// TIA Portal V16 program export: 1 tag tables, 0 data types, 0 data blocks, 1 code blocks (in call order from the OBs), 0 instance data blocks

VAR_GLOBAL   // PLC tag table "Electrical_interlock tag table"
   Stop AT %I0.0 : Bool;
   Start AT %I0.1 : Bool;
   Sistem AT %Q0.0 : Bool;
   btn_ileri AT %I0.2 : Bool;
   m_ileri AT %Q0.1 : Bool;
   btn_geri AT %I0.3 : Bool;
   m_geri AT %Q0.2 : Bool;
END_VAR

ORGANIZATION_BLOCK "Electrical_interlock"   // OB1, LAD, ProgramCycle
TITLE = "Main Program Sweep (Cycle)"
{ S7_Optimized_Access := 'TRUE' }
VERSION : 0.1
// stored: AutoNumber true, IsIECCheckEnabled false, SetENOAutomatically false
   VAR_INPUT
      Initial_Call : Bool;   // Initial call of this OB
      Remanence : Bool;   // =True, if remanent data are available
   END_VAR
BEGIN

REGION Network 1
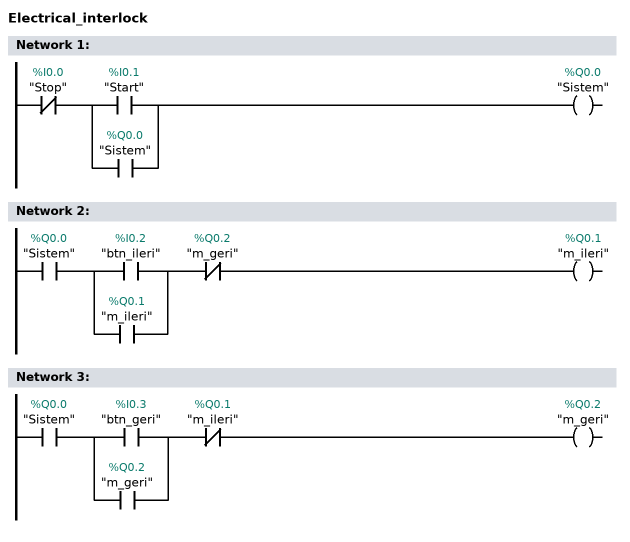
   RUNG wire#powerrail
      I_Contact( "Stop" )
      wire#w1
      Contact( "Start" )
      wire#w2
      Coil( "Sistem" )
   END_RUNG
   RUNG wire#w1
      Contact( "Sistem" )
   END_RUNG wire#w2
   // the same network as SCL:
   "Sistem" := NOT "Stop" AND ("Start" OR "Sistem");
END_REGION

REGION Network 2
   RUNG wire#powerrail
      Contact( "Sistem" )
      wire#w1
      Contact( "btn_ileri" )
      wire#w2
      I_Contact( "m_geri" )
      Coil( "m_ileri" )
   END_RUNG
   RUNG wire#w1
      Contact( "m_ileri" )
   END_RUNG wire#w2
   // the same network as SCL:
   "m_ileri" := "Sistem" AND ("btn_ileri" OR "m_ileri") AND NOT "m_geri";
END_REGION

REGION Network 3
   RUNG wire#powerrail
      Contact( "Sistem" )
      wire#w1
      Contact( "btn_geri" )
      wire#w2
      I_Contact( "m_ileri" )
      Coil( "m_geri" )
   END_RUNG
   RUNG wire#w1
      Contact( "m_geri" )
   END_RUNG wire#w2
   // the same network as SCL:
   "m_geri" := "Sistem" AND ("btn_geri" OR "m_geri") AND NOT "m_ileri";
END_REGION
END_ORGANIZATION_BLOCK
